FUNCTION_BLOCK FB_Output
VAR_INPUT
	bHandOverride:				BOOL;			//Wenn true kann der Ausgang auch im Handbetrieb geschrieben werden	
	fbSchrittbetrieb:			REFERENCE TO FB_Schrittbetrieb;
	bSendFalschePosError:		BOOL;
END_VAR
VAR_OUTPUT
	bFalschePos:				BOOL;
END_VAR
VAR
	bA_Output					AT%Q*: BOOL;
END_VAR

METHOD reset : BOOL
VAR_INPUT
END_VAR
VAR
	stSchrittEintrag:		ST_SchrittQueue;
END_VAR
stSchrittEintrag.fbOutput REF= THIS^;

//*************************************************************************************
IF		NOT Main.bE_Handbetrieb 
	AND NOT Main.bProgStop
	OR		bHandOverride

	OR		MAIN.bE_Handbetrieb							//Schritt vorwaerts im Handbetrieb
	AND		fbSchrittbetrieb.bAblaufFreigabe THEN
	
	//*************************************************************************************
	IF		 	bA_Output THEN	//Beim Wechsel des Ausgangs Bewegung in queue aufnehmen
		fbSchrittbetrieb.addToQueue(stSchrittEintrag);
	END_IF
	//*************************************************************************************
	
	bA_Output := FALSE;
	reset := TRUE;
END_IF
END_METHOD

METHOD set : BOOL
VAR_INPUT
END_VAR
VAR
	stSchrittEintrag:		ST_SchrittQueue;
END_VAR
stSchrittEintrag.fbOutput REF= THIS^;	
stSchrittEintrag.bGesetzt := TRUE;

//*************************************************************************************
IF		NOT Main.bE_Handbetrieb 
	AND NOT Main.bProgStop
	OR		bHandOverride

	OR		MAIN.bE_Handbetrieb							//Schritt vorwaerts im Handbetrieb
	AND		fbSchrittbetrieb.bAblaufFreigabe THEN
	
	//*************************************************************************************
	IF		NOT bA_Output THEN	//Beim Wechsel des Ausgangs Bewegung in queue aufnehmen
		fbSchrittbetrieb.addToQueue(stSchrittEintrag);
	END_IF
	//*************************************************************************************
	
	bA_Output := TRUE;
	set := TRUE;
END_IF
END_METHOD

END_FUNCTION_BLOCK

(* stored: Version 1.1.0.1, ProductVersion 3.1.4024.12
   POU FB_Output: Id {349d6daf-aa03-49e5-9785-0747744313b0}, SpecialFunc None
   Method reset: Id {3ef3f526-7e68-49de-a456-f609397e3f29}
   Method set: Id {da626f42-85ff-4793-89fb-bdfde239e8da} *)
